Fanuc TP program (LS listing): laser_test.ls

/PROG  LASER_TEST
/ATTR
OWNER		= MNEDITOR;
COMMENT		= "";
PROG_SIZE	= 508;
CREATE		= DATE 22-10-26  TIME 09:26:00;
MODIFIED	= DATE 22-10-26  TIME 09:33:44;
FILE_NAME	= ;
VERSION		= 0;
LINE_COUNT	= 3;
MEMORY_SIZE	= 868;
PROTECT		= READ_WRITE;
TCD:  STACK_SIZE	= 0,
      TASK_PRIORITY	= 50,
      TIME_SLICE	= 0,
      BUSY_LAMP_OFF	= 0,
      ABORT_REQUEST	= 0,
      PAUSE_REQUEST	= 0;
DEFAULT_GROUP	= 1,*,*,*,*;
CONTROL_CODE	= 00000000 00000000;
/APPL
/APPL

AUTO_SINGULARITY_HEADER;
  ENABLE_SINGULARITY_AVOIDANCE   : FALSE;
/MN
   1:  UFRAME_NUM=1 ;
   2:  UTOOL_NUM=6 ;
   3:J P[1] 100% FINE    ;
/POS
P[1]{
   GP1:
	UF : 1, UT : 6,		CONFIG : 'N U T, 0, 0, 0',
	X =     0.000  mm,	Y =     0.000  mm,	Z =   100.000  mm,
	W =     -.000 deg,	P =      .000 deg,	R =      .000 deg
};
/END
